TEXTLIST TextList
  1 = 'ESTADO DE LA ALARMA'
  2 = 'ABIERTO' | English: 'OPENED' | Spanish: 'ABIERTO'
  3 = 'ABRIENDO/\nCERRANDO' | English: 'OPENING/\nCLOSING' | Spanish: 'ABRIENDO/\nCERRANDO'
  4 = 'CERRADO' | English: 'CLOSED' | Spanish: 'CERRADO'
  5 = 'INTERRUPTOR' | English: 'SWITCH' | Spanish: 'INTERRUPTOR'
  6 = 'ALARMA' | English: 'ALARM' | Spanish: 'ALARMA'
  7 = 'CONFIGURACIÓN' | English: 'CONFIGURATION' | Spanish: 'CONFIGURACIÓN'
  0 = 'CONECTAR\n/DESCONECTAR \nPUERTA EMERGENCIA' | English: 'CONNECT/\nDISCONNECT\n EMERGENCY DOOR' | Spanish: 'CONECTAR/\nDESCONECTAR \nPUERTA EMERGENCIA'
  9 = 'PUERTA DE EMERGENCIA' | English: 'EMERGENCY DOOR' | Spanish: 'PUERTA DE EMERGENCIA'
   = ''
END_TEXTLIST

(* stored: Version 1.1.0.1, ProductVersion 3.1.4026.12
   TextList TextList: Id {78e8b958-b3c2-4b77-8900-a2aad21c6e3e} *)
